(* IEC 61131-3 sources: beckhoffAutomationInterface/ST/Shark/App/Shark/Programs, 13 files *)

(* ---- PRG_BronkhorstPressure.st ---- *)
(* Bronkhorst pressure controller application (Modbus needle valves).
   Creates Modbus hardware stack and controllers, then injects
   controller interfaces into PRG_PRESSURE_SENSOR via Configure(). *)
PROGRAM PRG_BronkhorstPressure
VAR
    // Modbus Hardware Stack
    fbModbusMaster       : ModbusRtuMasterV2_KL6x22B;
    fbNetworkCoordinator : FB_ModbusNetworkCoordinator;

    // Per-controller hardware
    aHardwareHandlers : ARRAY[1..GVL_PressureSystem.CONTROLLER_COUNT] OF FB_ModbusHardwareHandler;
    aDrivers          : ARRAY[1..GVL_PressureSystem.CONTROLLER_COUNT] OF FB_BronkhorstModbusAdapter;

    // Controllers
    aControllers : ARRAY[1..GVL_PressureSystem.CONTROLLER_COUNT] OF FB_BronkhorstController;
    aInterfaces  : ARRAY[1..GVL_PressureSystem.CONTROLLER_COUNT] OF I_Controller;

    bInitialized : BOOL := FALSE;
    i : INT;
END_VAR

    IF NOT bInitialized THEN
        _Init();
    END_IF

    // Execute Modbus communication
    fbModbusMaster();
    fbNetworkCoordinator.Execute();

    // Execute controllers
    FOR i := 1 TO GVL_PressureSystem.CONTROLLER_COUNT DO
        aControllers[i].Execute();
    END_FOR

METHOD PRIVATE _Init
    // PrecursorHot (slave 1)
    _InitController(
        eId           := E_PressureController.A_Side,
        nSlaveAddress := GVL_PressureSystem.MODBUS_FIRST_SLAVE_ADDRESS
    );

    // ReactantHot (slave 2)
    _InitController(
        eId           := E_PressureController.B_Side,
        nSlaveAddress := GVL_PressureSystem.MODBUS_FIRST_SLAVE_ADDRESS + 1
    );

    fbNetworkCoordinator.Init();

    // Inject controllers into pressure subsystem
    PRG_PRESSURE_SENSOR.Configure(aipCtrl := aInterfaces);

    bInitialized := TRUE;
END_METHOD

METHOD PRIVATE _InitController
VAR_INPUT
    eId           : E_PressureController;
    nSlaveAddress : BYTE;
END_VAR
VAR
    nIdx : INT;
END_VAR
    nIdx := eId;

    aHardwareHandlers[nIdx].Init(
        sInstanceName    := CONCAT('MODBUS_PRES_', TO_STRING(eId)),
        pModbusRtuMaster := ADR(fbModbusMaster),
        nSlaveAddress    := nSlaveAddress
    );
    aDrivers[nIdx].Init(
        sInstanceName      := CONCAT('DRV_', TO_STRING(eId)),
        nSlaveAddress      := nSlaveAddress,
        ipModbusComm       := aHardwareHandlers[nIdx],
        rFullScaleCapacity := GVL_PressureSystem.MAX_PRESSURE_CTRL_BAR,
        rMinimumValue      := GVL_PressureSystem.MIN_PRESSURE_CTRL_BAR
    );

    fbNetworkCoordinator.AddSlave(aDrivers[nIdx]);
    aDrivers[nIdx].SetPIDMode();

    aControllers[nIdx].Init(
        sInstanceName      := TO_STRING(eId),
        ipHardware         := aDrivers[nIdx],
        rMinValue          := GVL_PressureSystem.MIN_PRESSURE_CTRL_BAR,
        rMaxValue          := GVL_PressureSystem.MAX_PRESSURE_CTRL_BAR,
        bInverseControl    := TRUE,
        rBoundaryTolerance := GVL_PressureSystem.SETPOINT_TOLERANCE
    );

    aInterfaces[nIdx] := aControllers[nIdx];
END_METHOD

END_PROGRAM

(* ---- PRG_DIGITAL_INPUT.st ---- *)
(*
Digital Input Program - Shark System
Manages all digital inputs with centralized initialization.
*)
PROGRAM PRG_DIGITAL_INPUT
VAR
    // Subsystem and Manual Panel
    fbDigitalInputSubsystem : FB_DigitalInputSubsystem;
    fbManualPanel           : FB_DigitalInputManualPanel;

    // Hardware IO - Door Proximity Sensors
    IO_DoorLT            AT %I* : BOOL;
    IO_DoorLM            AT %I* : BOOL;
    IO_DoorLB            AT %I* : BOOL;
    IO_DoorRT            AT %I* : BOOL;
    IO_DoorRM            AT %I* : BOOL;
    IO_DoorRB            AT %I* : BOOL;
    IO_DoorBML           AT %I* : BOOL;
    IO_DoorBMR           AT %I* : BOOL;
    IO_DoorBMB           AT %I* : BOOL;

    // Safety-derived digital inputs (logical, not physical IO).
    // Updated each cycle from FB_SafetyManager via Configure()/I_SafetyStatus.
    _bHeaterVoltOn   : BOOL := FALSE;  // HETR_VOLT_ON — HeaterVoltagePresence
    _bSafetyOk       : BOOL := FALSE;  // SAFE_STO_ON  — safety state machine OK
    _bSafetyOverride : BOOL := TRUE;   // SAFE_OVERRIDE — no physical switch on Shark; always active

    // Safety status interface (injected via Configure)
    _ipSafety : I_SafetyStatus;

    // Function blocks and interfaces
    afbInputs : ARRAY[1..GVL_DIOConfig.DI_COUNT] OF FB_DigitalInput;
    aipInputs : ARRAY[1..GVL_DIOConfig.DI_COUNT] OF I_DigitalInput;

    bInitialized : BOOL := FALSE;
END_VAR

    IF NOT bInitialized THEN
        _Init();
    END_IF

    // Refresh safety-derived inputs before Execute() so subsystem reads fresh values each scan
    IF _ipSafety <> 0 THEN
        _bHeaterVoltOn := _ipSafety.HeaterVoltagePresence;
        _bSafetyOk     := _ipSafety.IsOk;
        // _bSafetyOverride stays TRUE — Shark has no physical override switch
    END_IF

    fbDigitalInputSubsystem.Execute();
    fbManualPanel(ipSubsystem := fbDigitalInputSubsystem, nMaxInput := GVL_DIOConfig.DI_COUNT);

METHOD PRIVATE _Init
VAR
    i : INT;
    apIO : ARRAY[1..GVL_DIOConfig.DI_COUNT] OF POINTER TO BOOL;
END_VAR
    // Build IO pointer mapping
    apIO[E_DigitalInputIdentifier.PRXS_DOOR_LT]    := ADR(IO_DoorLT);
    apIO[E_DigitalInputIdentifier.PRXS_DOOR_LM]    := ADR(IO_DoorLM);
    apIO[E_DigitalInputIdentifier.PRXS_DOOR_LB]    := ADR(IO_DoorLB);
    apIO[E_DigitalInputIdentifier.PRXS_DOOR_RT]    := ADR(IO_DoorRT);
    apIO[E_DigitalInputIdentifier.PRXS_DOOR_RM]    := ADR(IO_DoorRM);
    apIO[E_DigitalInputIdentifier.PRXS_DOOR_RB]    := ADR(IO_DoorRB);
    apIO[E_DigitalInputIdentifier.PRXS_DOOR_BML]   := ADR(IO_DoorBML);
    apIO[E_DigitalInputIdentifier.PRXS_DOOR_BMR]   := ADR(IO_DoorBMR);
    apIO[E_DigitalInputIdentifier.PRXS_DOOR_BMB]   := ADR(IO_DoorBMB);
    apIO[E_DigitalInputIdentifier.HETR_VOLT_ON]  := ADR(_bHeaterVoltOn);
    apIO[E_DigitalInputIdentifier.SAFE_STO_ON]   := ADR(_bSafetyOk);
    apIO[E_DigitalInputIdentifier.SAFE_OVERRIDE] := ADR(_bSafetyOverride);

    // Initialize all inputs using the mapping (all N.O. sensors, no inversion needed)
    FOR i := 1 TO GVL_DIOConfig.DI_COUNT DO
        IF apIO[i] <> 0 THEN
            afbInputs[i].Init(INT_TO_STRING(i), apIO[i]^);
            aipInputs[i] := afbInputs[i];
        END_IF
    END_FOR

    fbDigitalInputSubsystem.Init(aipInputs := aipInputs, nCount := GVL_DIOConfig.DI_COUNT);
    bInitialized := TRUE;
END_METHOD

METHOD PUBLIC Init : BOOL
VAR_INPUT
    ipSafety : I_SafetyStatus;
END_VAR
    IF ipSafety = 0 THEN
        Init := FALSE;
        RETURN;
    END_IF
    _ipSafety := ipSafety;
    Init := TRUE;
END_METHOD

END_PROGRAM

(* ---- PRG_DIGITAL_OUTPUT.st ---- *)
(*
Digital Output Program - Shark System
Manages all digital outputs with centralized initialization.
*)
PROGRAM PRG_DIGITAL_OUTPUT
VAR
    // Subsystem and Manual Panel
    fbDigitalOutputSubsystem : FB_DigitalOutputSubsystem;
    fbManualPanel            : FB_DigitalOutputManualPanel;

    // Hardware IO (Digital Outputs) - Signal Lights
    IO_SignalRed         AT %Q* : BOOL;
    IO_SignalYellow      AT %Q* : BOOL;
    IO_SignalGreen       AT %Q* : BOOL;

    // Hardware IO - Camera Lights
    IO_CameraLightTop    AT %Q* : BOOL;
    IO_CameraLightSide   AT %Q* : BOOL;

    // Hardware IO - Vacuum Pumps
    IO_ExhaustPump       AT %Q* : BOOL;
    IO_ChuckVacuumPump   AT %Q* : BOOL;

    // Hardware IO - Chiller
    IO_ChillerPower      AT %Q* : BOOL;

    // Hardware IO - Door Locks
    IO_DoorLockFL        AT %Q* : BOOL;
    IO_DoorLockFR        AT %Q* : BOOL;

    // Hardware IO - Heater Voltage Enable
    IO_HeaterVoltageOn   AT %Q* : BOOL;

    // Hardware IO - Solenoid Valve Outputs (consumed by PRG_VALVE)
    IO_ChuckLZ1          AT %Q* : BOOL;
    IO_ChuckLZ2          AT %Q* : BOOL;
    IO_ChuckLZ3          AT %Q* : BOOL;
    IO_ChuckVent         AT %Q* : BOOL;
    IO_ChuckWaterIn      AT %Q* : BOOL;
    IO_ChuckWaterOut     AT %Q* : BOOL;

    // Function blocks and interfaces
    afbOutputs : ARRAY[1..GVL_DIOConfig.DO_COUNT] OF FB_DigitalOutput;
    aipOutputs : ARRAY[1..GVL_DIOConfig.DO_COUNT] OF I_DigitalOutput;

    bInitialized : BOOL := FALSE;
END_VAR

    IF NOT bInitialized THEN
        _Init();
    END_IF

    fbDigitalOutputSubsystem.Execute();
    fbManualPanel(ipSubsystem := fbDigitalOutputSubsystem, nMaxOutput := GVL_DIOConfig.DO_COUNT);

METHOD PRIVATE _Init
VAR
    i : INT;
    apIO       : ARRAY[1..GVL_DIOConfig.DO_COUNT] OF POINTER TO BOOL;
    aSafeState : ARRAY[1..GVL_DIOConfig.DO_COUNT] OF BOOL;
END_VAR
    // ------------------------------------------------------------------
    // Safe states — applied by SetSafeState() on sequence abort / Halt().
    // Every output that is not listed here defaults to FALSE (de-energise).
    // SAFETY: door locks TRUE = stay locked; chiller TRUE = keep running.
    // ------------------------------------------------------------------
    aSafeState[E_DigitalOutputIdentifier.PUMP_AB_EXH]   := TRUE;
    aSafeState[E_DigitalOutputIdentifier.LGHT_SGN_GRN]  := FALSE; // Lights off
    aSafeState[E_DigitalOutputIdentifier.LGHT_SGN_RED]  := FALSE;
    aSafeState[E_DigitalOutputIdentifier.LGHT_SGN_YEL]  := FALSE;
    aSafeState[E_DigitalOutputIdentifier.LGHT_CMR_TOP]  := TRUE;
    aSafeState[E_DigitalOutputIdentifier.LGHT_CMR_SIDE] := TRUE;
    aSafeState[E_DigitalOutputIdentifier.CHIL_PWR]      := TRUE;  // SAFETY: chiller must keep running to protect hardware
    aSafeState[E_DigitalOutputIdentifier.LOCK_DOOR_FL]  := TRUE;  // SAFETY: doors stay locked on abort
    aSafeState[E_DigitalOutputIdentifier.LOCK_DOOR_FR]  := TRUE;  // SAFETY: doors stay locked on abort
    aSafeState[E_DigitalOutputIdentifier.VALV_CHK_LZ1]  := FALSE; // Chuck zone valves close
    aSafeState[E_DigitalOutputIdentifier.VALV_CHK_LZ2]  := FALSE;
    aSafeState[E_DigitalOutputIdentifier.VALV_CHK_LZ3]  := FALSE;
    aSafeState[E_DigitalOutputIdentifier.VALV_CHK_VENT] := FALSE; // Vent closes
    aSafeState[E_DigitalOutputIdentifier.VALV_CHK_WIN]  := FALSE; // Water valves close
    aSafeState[E_DigitalOutputIdentifier.VALV_CHK_WOUT] := FALSE;

    // Build IO pointer mapping
    apIO[E_DigitalOutputIdentifier.LGHT_SGN_RED]   := ADR(IO_SignalRed);
    apIO[E_DigitalOutputIdentifier.LGHT_SGN_YEL]   := ADR(IO_SignalYellow);
    apIO[E_DigitalOutputIdentifier.LGHT_SGN_GRN]   := ADR(IO_SignalGreen);
    apIO[E_DigitalOutputIdentifier.LGHT_CMR_TOP]   := ADR(IO_CameraLightTop);
    apIO[E_DigitalOutputIdentifier.LGHT_CMR_SIDE]  := ADR(IO_CameraLightSide);
    apIO[E_DigitalOutputIdentifier.PUMP_AB_EXH]    := ADR(IO_ExhaustPump);
    apIO[E_DigitalOutputIdentifier.PUMP_CHK_VAC]   := ADR(IO_ChuckVacuumPump);
    apIO[E_DigitalOutputIdentifier.CHIL_PWR]       := ADR(IO_ChillerPower);
    apIO[E_DigitalOutputIdentifier.LOCK_DOOR_FL]   := ADR(IO_DoorLockFL);
    apIO[E_DigitalOutputIdentifier.LOCK_DOOR_FR]   := ADR(IO_DoorLockFR);
    apIO[E_DigitalOutputIdentifier.VALV_CHK_LZ1]   := ADR(IO_ChuckLZ1);
    apIO[E_DigitalOutputIdentifier.VALV_CHK_LZ2]   := ADR(IO_ChuckLZ2);
    apIO[E_DigitalOutputIdentifier.VALV_CHK_LZ3]   := ADR(IO_ChuckLZ3);
    apIO[E_DigitalOutputIdentifier.VALV_CHK_VENT]  := ADR(IO_ChuckVent);
    apIO[E_DigitalOutputIdentifier.VALV_CHK_WIN]   := ADR(IO_ChuckWaterIn);
    apIO[E_DigitalOutputIdentifier.VALV_CHK_WOUT]  := ADR(IO_ChuckWaterOut);

    // Initialize all outputs using the mapping
    FOR i := 1 TO GVL_DIOConfig.DO_COUNT DO
        IF apIO[i] <> 0 THEN
            afbOutputs[i].Init(INT_TO_STRING(i), apIO[i]^, aSafeState[i]);
            aipOutputs[i] := afbOutputs[i];
        END_IF
    END_FOR

    fbDigitalOutputSubsystem.Init(aipOutputs := aipOutputs, nCount := GVL_DIOConfig.DO_COUNT);
    bInitialized := TRUE;
END_METHOD

END_PROGRAM

(* ---- PRG_HEAT_ZONE.st ---- *)
PROGRAM PRG_HEAT_ZONE
(*
Shark heater output wiring + temperature subsystem entry point.

  * 10 SSR outputs (one per channel) split across 8 zones.
  * Channel ordering MUST match PRG_TEMPERATURE_SENSOR's channel layout.
*)
VAR
    // --- Heater Digital Outputs (linked to EtherCAT process image) ---
    // HETR_HEAD   (channel 1)
    HEAD_Htr          AT %Q* : BOOL;
    // HETR_A_STR  (channel 2)
    A_STR_Htr         AT %Q* : BOOL;
    // HETR_A_CMB  (channel 3)
    A_CMB_Htr         AT %Q* : BOOL;
    // HETR_A_B1   (channel 4)
    A_B1_Htr          AT %Q* : BOOL;
    // HETR_A_B2   (channel 5)
    A_B2_Htr          AT %Q* : BOOL;
    // HETR_A_B3   (channel 6)
    A_B3_Htr          AT %Q* : BOOL;
    // HETR_B_STR  (channel 7)
    B_STR_Htr         AT %Q* : BOOL;
    // HETR_B_CMB  (channel 8)
    B_CMB_Htr         AT %Q* : BOOL;
    // HETR_B_B1   (channel 9)
    B_B1_Htr          AT %Q* : BOOL;
    // HETR_B_B2   (channel 10)
    B_B2_Htr          AT %Q* : BOOL;
    // HETR_B_B3   (channel 11)
    B_B3_Htr          AT %Q* : BOOL;
    // HETR_EXH    (channels 12..13)
    EXH_Htr           AT %Q* : BOOL;
    EXH_E2_Htr        AT %Q* : BOOL;
    // HETR_CHK    (channels 14..15)
    CHK_Htr           AT %Q* : BOOL;
    CHK_E2_Htr        AT %Q* : BOOL;

    // --- Heater Adapters ---
    afbElementHeaters : ARRAY[1..GVL_TemperatureZones.CHANNEL_MAX] OF FB_DigitalOutput;

    // --- Interface array consumed by FB_TemperatureSubsystem ---
    aipChannelHeaters : ARRAY[1..GVL_TemperatureZones.CHANNEL_MAX] OF I_DigitalOutput;

    // --- Application ---
    fbTemperatureSubsystem : FB_TemperatureSubsystem;
    fbManualPanel          : FB_TemperatureManualPanel;
    fbTuningPanel          : FB_BeckhoffTuningPanel;

    bInitialized : BOOL := FALSE;
END_VAR

    IF NOT bInitialized THEN
        _Init();
    END_IF

    // Run all zones and channels
    fbTemperatureSubsystem.Execute();

    // HMI Panels
    fbManualPanel(ipSubsystem := fbTemperatureSubsystem, nMaxZone := GVL_TemperatureZones.CONTROLLABLE_ZONE_MAX);
    fbTuningPanel(
        ipTunable := fbTemperatureSubsystem.GetTunable(
            eZone       := fbTuningPanel.iSelectedZoneIdx,
            nChannelIdx := fbTuningPanel.iSelectedChannelIdx,
            bWholeZone  := fbTuningPanel.bTuneWholeZone)
    );

METHOD PRIVATE _Init
    // Initialize channel heaters in channel-order (matches PRG_TEMPERATURE_SENSOR).
    _InitElement(1,  HEAD_Htr);
    _InitElement(2,  A_STR_Htr);
    _InitElement(3,  A_CMB_Htr);
    _InitElement(4,  A_B1_Htr);
    _InitElement(5,  A_B2_Htr);
    _InitElement(6,  A_B3_Htr);
    _InitElement(7,  B_STR_Htr);
    _InitElement(8,  B_CMB_Htr);
    _InitElement(9,  B_B1_Htr);
    _InitElement(10, B_B2_Htr);
    _InitElement(11, B_B3_Htr);
    _InitElement(12, EXH_Htr);
    _InitElement(13, EXH_E2_Htr);
    _InitElement(14, CHK_Htr);
    _InitElement(15, CHK_E2_Htr);

    // Initialize subsystem (sensors come from PRG_TEMPERATURE_SENSOR)
    bInitialized := fbTemperatureSubsystem.Init(
        aipChannelSensors := PRG_TEMPERATURE_SENSOR.aipChannelSensors,
        aipMonitorSensors := PRG_TEMPERATURE_SENSOR.aipMonitorSensors,
        aipChannelHeaters := aipChannelHeaters
    );
END_METHOD

METHOD PRIVATE _InitElement
VAR_INPUT
    nGlobalIdx : INT;
END_VAR
VAR_IN_OUT
    bOutput : BOOL;
END_VAR
    afbElementHeaters[nGlobalIdx].Init(
        sInstanceName := CONCAT('HEATER_E', TO_STRING(nGlobalIdx)),
        ipOutputRef   := bOutput
    );
    aipChannelHeaters[nGlobalIdx] := afbElementHeaters[nGlobalIdx];
END_METHOD

END_PROGRAM

(* ---- PRG_HUMIDITY_SENSOR.st ---- *)
(*
PRG_HUMIDITY_SENSOR — Ambient Humidity Sensor (Shark)

Manages the MDP5001_300_7E2119CA humidity channel from the Shark TH sensor pair.
Consumers read the scaled value via ipSensor.GetMeasurement().

The temperature channel of the same TH sensor is wired in PRG_TEMPERATURE_SENSOR
as E_TemperatureMonitorZone.SENS_CHAMBER.

Scaling constants are in GVL_HumiditySystem.
*)
PROGRAM PRG_HUMIDITY_SENSOR
VAR_INPUT
    // Hardware IO — linked to EtherCAT process image at %I* offset matching terminal position.
    // VAR_INPUT allows PRG_SIMULATION to write raw values for simulation mode.
    IO_Humid : T_Beckhoff_AmbientSensor;
END_VAR
VAR
    fbAdapter    : FB_AnalogInputAdapter;
    fbSensor     : FB_AnalogSensor;
    ipSensor     : I_Sensor;
    bInitialized : BOOL := FALSE;
END_VAR

    IF NOT bInitialized THEN
        _Init();
    END_IF

    fbAdapter.Execute();
    fbSensor.Execute();

METHOD PRIVATE _Init
    fbAdapter.Link(ADR(IO_Humid));
    fbSensor.Init(
        sInstanceName := 'AMBT_HUMID',
        ipRawInput    := fbAdapter,
        rRawMin       := GVL_HumiditySystem.AMBT_HUMID_RAW_MIN,
        rRawMax       := GVL_HumiditySystem.AMBT_HUMID_RAW_MAX,
        rScaledMin    := GVL_HumiditySystem.AMBT_HUMID_SCALED_MIN,
        rScaledMax    := GVL_HumiditySystem.AMBT_HUMID_SCALED_MAX
    );
    ipSensor     := fbSensor;
    bInitialized := TRUE;
END_METHOD

END_PROGRAM

(* ---- PRG_MFC.st ---- *)
PROGRAM PRG_MFC
VAR
    // Hardware IO - MFC Controllers (Bronkhorst EtherCAT)
    // Declared as VAR (not VAR_INPUT) so TwinCAT I/O linker exposes AT %I*/%Q*
    // members for EtherCAT PDO mapping. PRG_SIMULATION writes to these directly
    // via PRG_MFC.IO_MFC_*.MeasuredValue — this works identically for VAR.
    IO_MFC_Precursor : ST_BronkhorstController_IO;  // Range: 0-25 sccm
    IO_MFC_Reactant  : ST_BronkhorstController_IO;  // Range: 0-25 sccm
    IO_MFC_Inert     : ST_BronkhorstController_IO;  // Range: 0-500 sccm
END_VAR
VAR
    // Subsystem and Manual Panel
    fbFlowSubsystem : FB_FlowSubsystem;
    fbManualPanel   : FB_FlowManualPanel;

    // Adapters
    adapterPrecursor : FB_BronkhorstEtherCATAdapter;
    adapterReactant  : FB_BronkhorstEtherCATAdapter;
    adapterInert     : FB_BronkhorstEtherCATAdapter;

    // Controllers
    mfcPrecursor : FB_BronkhorstController;
    mfcReactant  : FB_BronkhorstController;
    mfcInert     : FB_BronkhorstController;

    bInitialized : BOOL := FALSE;
END_VAR

    IF NOT bInitialized THEN
        _Init();
    END_IF

    // Execute Controllers
    mfcPrecursor.Execute();
    mfcReactant.Execute();
    mfcInert.Execute();

    // Execute Subsystem (Error Aggregation)
    fbFlowSubsystem.Execute();

    // Manual Panel
    fbManualPanel(ipSubsystem := fbFlowSubsystem, nMaxZone := GVL_FlowSystem.FLOW_ZONE_COUNT);

METHOD PRIVATE _Init
VAR
    aipControllers : ARRAY[1..GVL_FlowSystem.FLOW_ZONE_COUNT] OF I_Controller;
END_VAR
    _InitMfc(
        eId          := E_MFCIdentifier.MFCT_A_01,
        stIo         := IO_MFC_Precursor,
        fbAdapter    := adapterPrecursor,
        fbController := mfcPrecursor,
        rMinValue    := GVL_FlowSystem.MIN_FLOW_PRECURSOR_SCCM,
        rMaxValue    := GVL_FlowSystem.MAX_FLOW_PRECURSOR_SCCM
    );
    _InitMfc(
        eId          := E_MFCIdentifier.MFCT_B_01,
        stIo         := IO_MFC_Reactant,
        fbAdapter    := adapterReactant,
        fbController := mfcReactant,
        rMinValue    := GVL_FlowSystem.MIN_FLOW_REACTANT_SCCM,
        rMaxValue    := GVL_FlowSystem.MAX_FLOW_REACTANT_SCCM
    );
    _InitMfc(
        eId          := E_MFCIdentifier.MFCT_IG_01,
        stIo         := IO_MFC_Inert,
        fbAdapter    := adapterInert,
        fbController := mfcInert,
        rMinValue    := GVL_FlowSystem.MIN_FLOW_INERT_SCCM,
        rMaxValue    := GVL_FlowSystem.MAX_FLOW_INERT_SCCM
    );

    // Subsystem Initialization
    aipControllers[E_MFCIdentifier.MFCT_A_01]  := mfcPrecursor;
    aipControllers[E_MFCIdentifier.MFCT_B_01]  := mfcReactant;
    aipControllers[E_MFCIdentifier.MFCT_IG_01] := mfcInert;

    fbFlowSubsystem.Init(aipControllers := aipControllers, nCount := GVL_FlowSystem.FLOW_ZONE_COUNT);
    bInitialized := TRUE;
END_METHOD

METHOD PRIVATE _InitMfc
VAR_INPUT
    eId       : E_MFCIdentifier;
    rMinValue : REAL;
    rMaxValue : REAL;
END_VAR
VAR_IN_OUT
    stIo         : ST_BronkhorstController_IO;
    fbAdapter    : FB_BronkhorstEtherCATAdapter;
    fbController : FB_BronkhorstController;
END_VAR
    fbAdapter.Link(
        refMeasuredValue     := stIo.MeasuredValue,
        refActualSetpoint    := stIo.ActualSetpoint,
        refValveOutput       := stIo.ValveOutput,
        refCommandedSetpoint := stIo.CommandedSetpoint,
        refControlByte       := stIo.ControlByte,
        refControlMode       := stIo.ControlMode,
        rMinValue            := REAL_TO_LREAL(rMinValue),
        rMaxValue            := REAL_TO_LREAL(rMaxValue)
    );
    fbController.Init(
        sInstanceName      := TO_STRING(eId),
        ipHardware         := fbAdapter,
        rMinValue          := rMinValue,
        rMaxValue          := rMaxValue,
        bInverseControl    := FALSE,
        rBoundaryTolerance := GVL_FlowSystem.SETPOINT_TOLERANCE
    );
END_METHOD

END_PROGRAM

(* ---- PRG_PRESSURE_SENSOR.st ---- *)
(*
Pressure Sensor Program - Shark System
Manages 4 analog pressure sensors with per-sensor scaling.
Bronkhorst pressure controllers are managed by PRG_BronkhorstPressure
and injected via Configure().

NOTE: PSNS_CHK_VAC has inverted physical mapping (higher raw = more vacuum = lower pressure).
      FB_AnalogSensor requires ascending ranges, so the reading is physically inverted.
      Consumers must compute: actual_pressure_bar = 1.0165 - sensor_reading
      TODO: Consider extending FB_AnalogSensor to support inverted scaling.
*)
PROGRAM PRG_PRESSURE_SENSOR
VAR
    // Hardware IO - Analog Pressure Sensors
    // Declared as VAR (not VAR_INPUT) so TwinCAT I/O linker exposes AT %I*/%Q*
    // members for EtherCAT PDO mapping. PRG_SIMULATION writes to these via
    // pointer/ADR — this works identically for VAR.
    IO_PressureSensors : ARRAY[1..GVL_PressureSystem.SENSOR_COUNT] OF T_Beckhoff_PressureSensor;
END_VAR
VAR
    // Subsystem and Manual Panel
    fbPressureSubsystem : FB_PressureSubsystem;
    fbManualPanel       : FB_PressureManualPanel;

    // Adapters and Sensors
    afbAdapters : ARRAY[1..GVL_PressureSystem.SENSOR_COUNT] OF FB_AnalogInputAdapter;
    afbSensors  : ARRAY[1..GVL_PressureSystem.SENSOR_COUNT] OF FB_AnalogSensor;

    // Interface arrays
    aipSensors     : ARRAY[1..GVL_PressureSystem.SENSOR_COUNT] OF I_Sensor;
    aipControllers : ARRAY[1..GVL_PressureSystem.CONTROLLER_COUNT] OF I_Controller;

    bConfigured     : BOOL := FALSE;
    bInitialized    : BOOL := FALSE;
    _bNotConfiguredLogged : BOOL := FALSE;
    i : INT;
END_VAR

    IF NOT bConfigured THEN
        IF NOT _bNotConfiguredLogged THEN
            GVL_ErrorLogger.Logger.LogError(
                sSource  := 'PRG_PRESSURE_SENSOR',
                eErrorId := E_ErrorId.ERR_GEN_NOT_CONFIGURED,
                sContext := 'PRG_PRESSURE_SENSOR executed before Configure(); pressure sensors will not run'
            );
            _bNotConfiguredLogged := TRUE;
        END_IF
        RETURN;
    END_IF

    IF NOT bInitialized THEN
        _Init();
    END_IF

    // Execute adapters and sensors
    FOR i := 1 TO GVL_PressureSystem.SENSOR_COUNT DO
        afbAdapters[i].Execute();
        afbSensors[i].Execute();
    END_FOR

    // Execute subsystem (error aggregation)
    fbPressureSubsystem.Execute();
    fbManualPanel(ipSubsystem := fbPressureSubsystem, nMaxSensor := GVL_PressureSystem.SENSOR_COUNT, nMaxCtrl := GVL_PressureSystem.CONTROLLER_COUNT);

    // Dependency injection - accepts controller interfaces from PRG_BronkhorstPressure
METHOD PUBLIC Configure
VAR_INPUT
    aipCtrl : ARRAY[1..GVL_PressureSystem.CONTROLLER_COUNT] OF I_Controller;
END_VAR
VAR
    iLocal : INT;
END_VAR
    IF bConfigured THEN RETURN;
    END_IF

    FOR iLocal := 1 TO GVL_PressureSystem.CONTROLLER_COUNT DO
        aipControllers[iLocal] := aipCtrl[iLocal];
    END_FOR

    bConfigured := TRUE;
END_METHOD

METHOD PRIVATE _Init
VAR
    eId : E_PressureSensorIdentifier;
END_VAR
    // PSNS_A_DST: A-side Distributor [0-3 bar]
    _InitSensor(
        eId       := E_PressureSensorIdentifier.PSNS_A_DST,
        rRawMin   := GVL_PressureSystem.PSNS_A_DST_RAW_MIN,
        rRawMax   := GVL_PressureSystem.PSNS_A_DST_RAW_MAX,
        rScaledMin := GVL_PressureSystem.PSNS_A_DST_SCALED_MIN,
        rScaledMax := GVL_PressureSystem.PSNS_A_DST_SCALED_MAX
    );

    // PSNS_B_DST: B-side Distributor [0-3 bar]
    _InitSensor(
        eId       := E_PressureSensorIdentifier.PSNS_B_DST,
        rRawMin   := GVL_PressureSystem.PSNS_B_DST_RAW_MIN,
        rRawMax   := GVL_PressureSystem.PSNS_B_DST_RAW_MAX,
        rScaledMin := GVL_PressureSystem.PSNS_B_DST_SCALED_MIN,
        rScaledMax := GVL_PressureSystem.PSNS_B_DST_SCALED_MAX
    );

    // PSNS_AB_EXH: Exhaust Vacuum [0-1 bar]
    _InitSensor(
        eId       := E_PressureSensorIdentifier.PSNS_AB_EXH,
        rRawMin   := GVL_PressureSystem.PSNS_AB_EXH_RAW_MIN,
        rRawMax   := GVL_PressureSystem.PSNS_AB_EXH_RAW_MAX,
        rScaledMin := GVL_PressureSystem.PSNS_AB_EXH_SCALED_MIN,
        rScaledMax := GVL_PressureSystem.PSNS_AB_EXH_SCALED_MAX
    );

    // PSNS_CHK_VAC: Chuck Vacuum [inverted: see NOTE above]
    _InitSensor(
        eId       := E_PressureSensorIdentifier.PSNS_CHK_VAC,
        rRawMin   := GVL_PressureSystem.PSNS_CHK_VAC_RAW_MIN,
        rRawMax   := GVL_PressureSystem.PSNS_CHK_VAC_RAW_MAX,
        rScaledMin := GVL_PressureSystem.PSNS_CHK_VAC_SCALED_MIN,
        rScaledMax := GVL_PressureSystem.PSNS_CHK_VAC_SCALED_MAX
    );

    // Initialize subsystem with sensors + injected controllers
    fbPressureSubsystem.Init(aipSensors := aipSensors, nSensorCount := GVL_PressureSystem.SENSOR_COUNT, aipControllers := aipControllers, nControllerCount := GVL_PressureSystem.CONTROLLER_COUNT);
    bInitialized := TRUE;
END_METHOD

METHOD PRIVATE _InitSensor
VAR_INPUT
    eId        : E_PressureSensorIdentifier;
    rRawMin    : LREAL;
    rRawMax    : LREAL;
    rScaledMin : LREAL;
    rScaledMax : LREAL;
END_VAR
VAR
    nIdx : INT;
END_VAR
    nIdx := eId;

    afbAdapters[nIdx].Link(ADR(IO_PressureSensors[nIdx]));
    afbSensors[nIdx].Init(
        sInstanceName := TO_STRING(eId),
        ipRawInput    := afbAdapters[nIdx],
        rRawMin       := rRawMin,
        rRawMax       := rRawMax,
        rScaledMin    := rScaledMin,
        rScaledMax    := rScaledMax
    );
    aipSensors[nIdx] := afbSensors[nIdx];
END_METHOD

END_PROGRAM

(* ---- PRG_Sequence.st ---- *)
// Runs the sequence orchestrator and the sequence tester side-by-side.
// Tester is wired to the orchestrator during Configure — no separate PRG_SequenceTester needed.
PROGRAM PRG_Sequence
VAR
    fbOrchestrator : FB_SequenceOrchestrator;
    fbTester       : FB_SequenceTester;
END_VAR

    fbOrchestrator();
    fbTester();

END_PROGRAM

METHOD PUBLIC Configure : BOOL
VAR_INPUT
    ipProvider : I_HardwareProvider;
END_VAR
    Configure := fbOrchestrator.Configure(ipProvider := ipProvider);
    fbTester.Configure(refOrchestrator := fbOrchestrator);
END_METHOD

METHOD PUBLIC GetStatus : ST_SequenceStatus
    GetStatus := fbOrchestrator.GetStatus();
END_METHOD

(* ---- PRG_SIMULATION.st ---- *)
(*
PRG_SIMULATION — I/O Hijacking Simulator for Shark Machine

Writes directly to the bottom-most layer:
  - Beckhoff sensor structs (T_Beckhoff_TempSensor_*, T_Beckhoff_PressureSensor)
    via raw INT pointer writes at offset 2.
  - Bronkhorst Modbus adapters via InjectMeasuredValue() (overwrites the polled
    rMeasuredValue, symmetric to PRO's EtherCAT IO struct hijack).
  - EtherCAT MFC IO fields (ST_BronkhorstController_IO.MeasuredValue) directly.

Everything above (FB_AnalogInputAdapter → FB_AnalogSensor → controllers → UI)
works naturally without knowing it's simulated.

Shark has 10 heater zones (no B-side zones 7-11), 4 pressure sensors,
3 EtherCAT MFCs, and Modbus-based pressure controllers.

PHYSICS ENGINE:
  FB_GasPhysicsSimulator reads valve states + pump state from the previous cycle,
  computes CM/HM pressures and MFC flow, and outputs are written to sensor IO.
*)
PROGRAM PRG_SIMULATION
VAR
    // Hardware provider — injected via Configure() from PRG_SHARK
    _ipProvider  : I_HardwareProvider;
    _bConfigured : BOOL := FALSE;

    // Gas system physics — pressure + flow for both sides
    fbGasPhysics : FB_GasPhysicsSimulator;

    // Temperature physics — one per channel channel
    aSimHeaters : ARRAY[1..GVL_TemperatureZones.CHANNEL_MAX] OF FB_SimulateHeaterZone;

    // Inert MFC simulation (not part of gas side physics)
    fbSimMFC_Inert : FB_SimulateAnalogActuator;

    // Working
    bInitialized : BOOL := FALSE;
END_VAR

IF NOT GVL_Simulation.bActive THEN
    RETURN;
END_IF

IF NOT bInitialized THEN
    _Init();
END_IF

// =============================================================================
// 0. SAFETY — Force safe state so subsystems can run
// =============================================================================
GVL_Safety.SafetyOk := TRUE;
GVL_Safety.HeaterVoltage := 230.0;

// =============================================================================
// 1. TEMPERATURE — Write directly to T_Beckhoff_TempSensor structs (no provider)
// =============================================================================
_SimulateTemperature();

// =============================================================================
// 2. GAS PHYSICS + PRESSURE + MFC (requires provider — first cycle is a no-op,
//    _Init atmospheric seed is preserved until provider is wired on cycle 2)
// =============================================================================
IF _bConfigured THEN
    _SimulateGasPhysics();
    _SimulatePressureSensors();
    _SimulateMFCs();
    _SimulateModbusPressureControllers();
END_IF

// =============================================================================
// CONFIGURATION
// =============================================================================

METHOD PUBLIC Configure
VAR_INPUT
    ipProvider : I_HardwareProvider;
END_VAR
    _ipProvider  := ipProvider;
    _bConfigured := _ipProvider <> 0;
END_METHOD

// =============================================================================
// INITIALIZATION
// =============================================================================

METHOD PRIVATE _Init
VAR
    iZone      : INT;
    e          : INT;
    nGlobalIdx : INT;
    nCount     : INT;
    iSensor    : INT;
END_VAR
    // Temperature: init physics for every channel of every populated zone
    nGlobalIdx := 0;
    FOR iZone := 1 TO GVL_TemperatureZones.CONTROLLABLE_ZONE_MAX DO
        nCount := GVL_TemperatureZoneConfig.ZONE_CONFIG[iZone].nChannelCount;
        FOR e := 1 TO nCount DO
            nGlobalIdx := nGlobalIdx + 1;
            IF nGlobalIdx > GVL_TemperatureZones.CHANNEL_MAX THEN EXIT; END_IF
            IF GVL_TemperatureZoneConfig.ZONE_CONFIG[iZone].bPopulated THEN
                aSimHeaters[nGlobalIdx].Init(
                    rAmbient     := GVL_SimulationConfig.AMBIENT_TEMP,
                    rHeatingRate := GVL_SimulationConfig.HEATING_RATE,
                    rCoolingRate := GVL_SimulationConfig.COOLING_RATE,
                    rMaxTemp     := LREAL_TO_REAL(GVL_TemperatureZoneConfig.ZONE_CONFIG[iZone].rMaxSetpoint)
                );
            END_IF
        END_FOR
    END_FOR

    // Pressure: seed sensors with atmospheric so first-cycle reads are valid
    FOR iSensor := 1 TO GVL_PressureSystem.SENSOR_COUNT DO
        _WriteSensorRaw(
            ADR(PRG_PRESSURE_SENSOR.IO_PressureSensors[iSensor]),
            _PressureToRaw(GVL_SimulationConfig.ATMOSPHERIC_PRESSURE, iSensor));
    END_FOR

    bInitialized := TRUE;
END_METHOD

// =============================================================================
// TEMPERATURE SIMULATION
// =============================================================================

METHOD PRIVATE _SimulateTemperature
    // Channel 1: HETR_HEAD
    _SimulateElement(1,  PRG_HEAT_ZONE.HEAD_Htr,
        ADR(PRG_TEMPERATURE_SENSOR.HEAD_A),
        ADR(PRG_TEMPERATURE_SENSOR.HEAD_B));

    // Channels 2-6: A-side STR/CMB/B1/B2/B3
    _SimulateElement(2,  PRG_HEAT_ZONE.A_STR_Htr,
        ADR(PRG_TEMPERATURE_SENSOR.A_STR_A),
        ADR(PRG_TEMPERATURE_SENSOR.A_STR_B));
    _SimulateElement(3,  PRG_HEAT_ZONE.A_CMB_Htr,
        ADR(PRG_TEMPERATURE_SENSOR.A_CMB_A),
        ADR(PRG_TEMPERATURE_SENSOR.A_CMB_B));
    _SimulateElement(4,  PRG_HEAT_ZONE.A_B1_Htr,
        ADR(PRG_TEMPERATURE_SENSOR.A_B1_A),
        ADR(PRG_TEMPERATURE_SENSOR.A_B1_B));
    _SimulateElement(5,  PRG_HEAT_ZONE.A_B2_Htr,
        ADR(PRG_TEMPERATURE_SENSOR.A_B2_A),
        ADR(PRG_TEMPERATURE_SENSOR.A_B2_B));
    _SimulateElement(6,  PRG_HEAT_ZONE.A_B3_Htr,
        ADR(PRG_TEMPERATURE_SENSOR.A_B3_A),
        ADR(PRG_TEMPERATURE_SENSOR.A_B3_B));

    // Channels 7-11: B-side STR/CMB/B1/B2/B3
    _SimulateElement(7,  PRG_HEAT_ZONE.B_STR_Htr,
        ADR(PRG_TEMPERATURE_SENSOR.B_STR_A),
        ADR(PRG_TEMPERATURE_SENSOR.B_STR_B));
    _SimulateElement(8,  PRG_HEAT_ZONE.B_CMB_Htr,
        ADR(PRG_TEMPERATURE_SENSOR.B_CMB_A),
        ADR(PRG_TEMPERATURE_SENSOR.B_CMB_B));
    _SimulateElement(9,  PRG_HEAT_ZONE.B_B1_Htr,
        ADR(PRG_TEMPERATURE_SENSOR.B_B1_A),
        ADR(PRG_TEMPERATURE_SENSOR.B_B1_B));
    _SimulateElement(10, PRG_HEAT_ZONE.B_B2_Htr,
        ADR(PRG_TEMPERATURE_SENSOR.B_B2_A),
        ADR(PRG_TEMPERATURE_SENSOR.B_B2_B));
    _SimulateElement(11, PRG_HEAT_ZONE.B_B3_Htr,
        ADR(PRG_TEMPERATURE_SENSOR.B_B3_A),
        ADR(PRG_TEMPERATURE_SENSOR.B_B3_B));

    // Channels 12-13: HETR_EXH (inner + outer)
    _SimulateElement(12, PRG_HEAT_ZONE.EXH_Htr,
        ADR(PRG_TEMPERATURE_SENSOR.EXH_IN_A),
        ADR(PRG_TEMPERATURE_SENSOR.EXH_IN_B));
    _SimulateElement(13, PRG_HEAT_ZONE.EXH_E2_Htr,
        ADR(PRG_TEMPERATURE_SENSOR.EXH_OUT_A),
        ADR(PRG_TEMPERATURE_SENSOR.EXH_OUT_B));

    // Channels 14-15: HETR_CHK (inner + outer, single sensor per channel)
    _SimulateElement(14, PRG_HEAT_ZONE.CHK_Htr,
        ADR(PRG_TEMPERATURE_SENSOR.CHK_IN_A),
        0);
    _SimulateElement(15, PRG_HEAT_ZONE.CHK_E2_Htr,
        ADR(PRG_TEMPERATURE_SENSOR.CHK_OUT_A),
        0);
END_METHOD

// =============================================================================
// GAS PHYSICS SIMULATION
// =============================================================================

(* Read valve/pump states from previous cycle, run physics, produce pressures + flows *)
METHOD PRIVATE _SimulateGasPhysics
VAR
    ipOutput : I_DigitalOutput;
    ipValve  : I_Valve;
END_VAR
    // System state — null-safe (provider may transiently return 0 during init)
    ipOutput := _ipProvider.GetExhaustPump();
    fbGasPhysics.bPumpOn := (ipOutput <> 0) AND_THEN ipOutput.GetOutput();
    ipValve := _ipProvider.GetExhaustVacuumIsoValve();
    fbGasPhysics.bExhaustVacuumIsoOpen := (ipValve <> 0) AND_THEN ipValve.IsOpen();

    // Per-side valve + controller states
    fbGasPhysics.stASide := _ReadSideState(E_GasSide.A_SIDE);
    fbGasPhysics.stBSide := _ReadSideState(E_GasSide.B_SIDE);

    fbGasPhysics.Execute();
END_METHOD

(* Build ST_GasSideState from domain getters — eliminates A/B duplication.
   All provider calls are null-safe via AND_THEN to tolerate partial init. *)
METHOD PRIVATE _ReadSideState : ST_GasSideState
VAR_INPUT
    eSide : E_GasSide;
END_VAR
VAR
    ipValve  : I_Valve;
    ipCtrl   : I_Controller;
    stStatus : ST_ControllerStatus;
END_VAR
    // Gas input
    ipValve := _ipProvider.GetGasIsoValve(eSide, 1);
    _ReadSideState.bGasIsoOpen      := (ipValve <> 0) AND_THEN ipValve.IsOpen();
    ipCtrl := _ipProvider.GetMFCController(eSide);
    IF ipCtrl <> 0 THEN
        stStatus := ipCtrl.GetStatus();
        _ReadSideState.rMFCSetpoint := stStatus.rSetpoint;
    END_IF

    // Cold manifold
    ipValve := _ipProvider.GetCMBubblerValve(eSide, 1);
    _ReadSideState.bCMBubbler1Open  := (ipValve <> 0) AND_THEN ipValve.IsOpen();
    ipValve := _ipProvider.GetCMBubblerValve(eSide, 2);
    _ReadSideState.bCMBubbler2Open  := (ipValve <> 0) AND_THEN ipValve.IsOpen();
    ipValve := _ipProvider.GetCMBubblerValve(eSide, 3);
    _ReadSideState.bCMBubbler3Open  := (ipValve <> 0) AND_THEN ipValve.IsOpen();
    ipValve := _ipProvider.GetCMPurgeValve(eSide);
    _ReadSideState.bCMPurgeOpen     := (ipValve <> 0) AND_THEN ipValve.IsOpen();
    ipValve := _ipProvider.GetCMVacuumIsoValve(eSide);
    _ReadSideState.bCMVacuumIsoOpen := (ipValve <> 0) AND_THEN ipValve.IsOpen();

    // Hot manifold
    ipValve := _ipProvider.GetHMBubblerValve(eSide, 1);
    _ReadSideState.bHMBubbler1Open  := (ipValve <> 0) AND_THEN ipValve.IsOpen();
    ipValve := _ipProvider.GetHMBubblerValve(eSide, 2);
    _ReadSideState.bHMBubbler2Open  := (ipValve <> 0) AND_THEN ipValve.IsOpen();
    ipValve := _ipProvider.GetHMBubblerValve(eSide, 3);
    _ReadSideState.bHMBubbler3Open  := (ipValve <> 0) AND_THEN ipValve.IsOpen();
    ipValve := _ipProvider.GetHMPurgeValve(eSide);
    _ReadSideState.bHMPurgeOpen     := (ipValve <> 0) AND_THEN ipValve.IsOpen();
    ipValve := _ipProvider.GetHMVacuumIsoValve(eSide);
    _ReadSideState.bHMVacuumIsoOpen := (ipValve <> 0) AND_THEN ipValve.IsOpen();

    // Output
    ipValve := _ipProvider.GetNozzleIsoValve(eSide);
    _ReadSideState.bNozzleIsoOpen   := (ipValve <> 0) AND_THEN ipValve.IsOpen();
    ipCtrl := _ipProvider.GetPressureController(eSide);
    IF ipCtrl <> 0 THEN
        stStatus := ipCtrl.GetStatus();
        _ReadSideState.rPCVSetpoint := stStatus.rSetpoint;
    END_IF
END_METHOD

// =============================================================================
// PRESSURE SENSOR SIMULATION
// =============================================================================

(* Write physics-computed pressures to analog pressure sensor raw IO *)
METHOD PRIVATE _SimulatePressureSensors
    // A-side distributor (cold manifold) pressure
    _WriteSensorRaw(
        ADR(PRG_PRESSURE_SENSOR.IO_PressureSensors[E_PressureSensorIdentifier.PSNS_A_DST]),
        _PressureToRaw(LREAL_TO_REAL(fbGasPhysics.stASideOut.rCMPressure), E_PressureSensorIdentifier.PSNS_A_DST));

    // B-side distributor (cold manifold) pressure
    _WriteSensorRaw(
        ADR(PRG_PRESSURE_SENSOR.IO_PressureSensors[E_PressureSensorIdentifier.PSNS_B_DST]),
        _PressureToRaw(LREAL_TO_REAL(fbGasPhysics.stBSideOut.rCMPressure), E_PressureSensorIdentifier.PSNS_B_DST));

    // Exhaust vacuum pressure
    _WriteSensorRaw(
        ADR(PRG_PRESSURE_SENSOR.IO_PressureSensors[E_PressureSensorIdentifier.PSNS_AB_EXH]),
        _PressureToRaw(LREAL_TO_REAL(fbGasPhysics.rExhaustPressure), E_PressureSensorIdentifier.PSNS_AB_EXH));

    // Chuck vacuum pressure � driven by dedicated PUMP_CHK_VAC state
    _WriteSensorRaw(
        ADR(PRG_PRESSURE_SENSOR.IO_PressureSensors[E_PressureSensorIdentifier.PSNS_CHK_VAC]),
        _PressureToRaw(_GetChuckVacuumPressure(), E_PressureSensorIdentifier.PSNS_CHK_VAC));
END_METHOD

// =============================================================================
// MFC SIMULATION
// =============================================================================

(* Write physics-computed MFC flow to EtherCAT IO. Inert MFC uses simple ramp.
   Direct assignment to VAR members of another PROGRAM is prohibited (C0037),
   so pointer writes are used — identical pattern to _WriteSensorRaw.
   MeasuredValue is UINT (0-32000 raw counts); convert from engineering units. *)
METHOD PRIVATE _SimulateMFCs
VAR
    _pUINT : POINTER TO UINT;
END_VAR
    // A-side Precursor — from gas physics
    _pUINT := ADR(PRG_MFC.IO_MFC_Precursor.MeasuredValue);
    _pUINT^ := WORD_TO_UINT(F_EngineeringToRawCounts(
        fbGasPhysics.stASideOut.rMFCActual,
        REAL_TO_LREAL(GVL_FlowSystem.MIN_FLOW_PRECURSOR_SCCM),
        REAL_TO_LREAL(GVL_FlowSystem.MAX_FLOW_PRECURSOR_SCCM), 32000));

    // B-side Reactant — from gas physics
    _pUINT := ADR(PRG_MFC.IO_MFC_Reactant.MeasuredValue);
    _pUINT^ := WORD_TO_UINT(F_EngineeringToRawCounts(
        fbGasPhysics.stBSideOut.rMFCActual,
        REAL_TO_LREAL(GVL_FlowSystem.MIN_FLOW_REACTANT_SCCM),
        REAL_TO_LREAL(GVL_FlowSystem.MAX_FLOW_REACTANT_SCCM), 32000));

    // Inert — independent, simple ramp (not part of gas side physics)
    // CommandedSetpoint is UINT; convert to engineering units for the ramp simulator.
    fbSimMFC_Inert(
        rSetpoint := LREAL_TO_REAL(F_RawCountsToEngineering(
            PRG_MFC.IO_MFC_Inert.CommandedSetpoint,
            REAL_TO_LREAL(GVL_FlowSystem.MIN_FLOW_INERT_SCCM),
            REAL_TO_LREAL(GVL_FlowSystem.MAX_FLOW_INERT_SCCM), 32000)),
        rRampRate := GVL_SimulationConfig.MFC_RAMP_RATE
    );
    _pUINT := ADR(PRG_MFC.IO_MFC_Inert.MeasuredValue);
    _pUINT^ := WORD_TO_UINT(F_EngineeringToRawCounts(
        REAL_TO_LREAL(fbSimMFC_Inert.rActualFeedback),
        REAL_TO_LREAL(GVL_FlowSystem.MIN_FLOW_INERT_SCCM),
        REAL_TO_LREAL(GVL_FlowSystem.MAX_FLOW_INERT_SCCM), 32000));
END_METHOD

// =============================================================================
// MODBUS PRESSURE CONTROLLER SIMULATION
// =============================================================================

(* Inject physics-computed HM pressure into Modbus pressure controller adapters.
   Symmetric to PRO's EtherCAT path which writes IO_CtrlASide.MeasuredValue directly:
   InjectMeasuredValue() overwrites the value that Modbus polling would normally update. *)
METHOD PRIVATE _SimulateModbusPressureControllers
    PRG_BronkhorstPressure.aDrivers[E_PressureController.A_Side].InjectMeasuredValue(fbGasPhysics.stASideOut.rHMPressure);
    PRG_BronkhorstPressure.aDrivers[E_PressureController.B_Side].InjectMeasuredValue(fbGasPhysics.stBSideOut.rHMPressure);
END_METHOD

// =============================================================================
// PRIVATE HELPERS
// =============================================================================

(* Run physics for one channel and write result to both A+B redundant sensor channels *)
METHOD PRIVATE _SimulateElement
VAR_INPUT
    nGlobalIdx : INT;
    bHeaterOn  : BOOL;
    pSensorA   : POINTER TO BYTE;
    pSensorB   : POINTER TO BYTE;
END_VAR
VAR
    nRawValue : INT;
END_VAR
    IF nGlobalIdx < 1 OR nGlobalIdx > GVL_TemperatureZones.CHANNEL_MAX THEN RETURN; END_IF
    aSimHeaters[nGlobalIdx](bHeaterOn := bHeaterOn);
    nRawValue := _TempToRaw(aSimHeaters[nGlobalIdx].rCurrentTemp);
    _WriteSensorRaw(pSensorA, nRawValue);
    _WriteSensorRaw(pSensorB, nRawValue);
END_METHOD

(* Return the simulated chuck vacuum pressure based on PUMP_CHK_VAC output state.
   PUMP_CHK_VAC is the dedicated chuck vacuum pump (not shared with exhaust).
   Pump ON  ? vacuum achieved: CHUCK_VACUUM_PRESSURE (0.01 bar)
   Pump OFF ? atmospheric: ATMOSPHERIC_PRESSURE (1.0 bar) *)
METHOD PRIVATE _GetChuckVacuumPressure : REAL
VAR
    ipPump : I_DigitalOutput;
END_VAR
    ipPump := _ipProvider.GetDigitalOutput(E_DigitalOutputIdentifier.PUMP_CHK_VAC);
    _GetChuckVacuumPressure := SEL(
        (ipPump <> 0) AND_THEN ipPump.GetOutput(),
        GVL_SimulationConfig.ATMOSPHERIC_PRESSURE,
        GVL_SimulationConfig.CHUCK_VACUUM_PRESSURE);
END_METHOD

(* Convert °C to Beckhoff EL32xx raw INT. Scale: 0.1°C per count → 25.0°C = 250 *)
METHOD PRIVATE _TempToRaw : INT
VAR_INPUT
    rTempC : REAL;
END_VAR
    _TempToRaw := REAL_TO_INT(rTempC / LREAL_TO_REAL(GVL_TemperatureSystem.SCALE_BECKHOFF_TEMP));
END_METHOD

(* Convert bar to Beckhoff EL3048 raw INT using per-sensor scaling from GVL_PressureSystem.
   Each sensor has different raw/scaled ranges. *)
METHOD PRIVATE _PressureToRaw : INT
VAR_INPUT
    rBar     : REAL;
    nSensor  : INT;
END_VAR
    CASE nSensor OF
    1: // PSNS_A_DST: 0-30518 raw → 0-3 bar
        _PressureToRaw := F_ScaleRealToInt(rBar,
            LREAL_TO_REAL(GVL_PressureSystem.PSNS_A_DST_SCALED_MIN),
            LREAL_TO_REAL(GVL_PressureSystem.PSNS_A_DST_SCALED_MAX),
            LREAL_TO_INT(GVL_PressureSystem.PSNS_A_DST_RAW_MIN),
            LREAL_TO_INT(GVL_PressureSystem.PSNS_A_DST_RAW_MAX));
    2: // PSNS_B_DST: 0-30518 raw → 0-3 bar
        _PressureToRaw := F_ScaleRealToInt(rBar,
            LREAL_TO_REAL(GVL_PressureSystem.PSNS_B_DST_SCALED_MIN),
            LREAL_TO_REAL(GVL_PressureSystem.PSNS_B_DST_SCALED_MAX),
            LREAL_TO_INT(GVL_PressureSystem.PSNS_B_DST_RAW_MIN),
            LREAL_TO_INT(GVL_PressureSystem.PSNS_B_DST_RAW_MAX));
    3: // PSNS_AB_EXH: 0-30518 raw → 0-1 bar
        _PressureToRaw := F_ScaleRealToInt(rBar,
            LREAL_TO_REAL(GVL_PressureSystem.PSNS_AB_EXH_SCALED_MIN),
            LREAL_TO_REAL(GVL_PressureSystem.PSNS_AB_EXH_SCALED_MAX),
            LREAL_TO_INT(GVL_PressureSystem.PSNS_AB_EXH_RAW_MIN),
            LREAL_TO_INT(GVL_PressureSystem.PSNS_AB_EXH_RAW_MAX));
    4: // PSNS_CHK_VAC: 3052-15259 raw → 0.00325-1.01325 bar (inverted physical)
        _PressureToRaw := F_ScaleRealToInt(rBar,
            LREAL_TO_REAL(GVL_PressureSystem.PSNS_CHK_VAC_SCALED_MIN),
            LREAL_TO_REAL(GVL_PressureSystem.PSNS_CHK_VAC_SCALED_MAX),
            LREAL_TO_INT(GVL_PressureSystem.PSNS_CHK_VAC_RAW_MIN),
            LREAL_TO_INT(GVL_PressureSystem.PSNS_CHK_VAC_RAW_MAX));
    END_CASE
END_METHOD

(* Write raw INT to a Beckhoff sensor struct at offset 2.
   All EL3xxx structs share the same memory layout:
   Offset 0-1: Status WORD, Offset 2-3: Value INT.
   This matches how FB_AnalogInputAdapter reads — same offset, reverse direction. *)
METHOD PRIVATE _WriteSensorRaw
VAR_INPUT
    pSensor   : POINTER TO BYTE;
    nRawValue : INT;
END_VAR
VAR
    pValue : POINTER TO INT;
END_VAR
    IF pSensor = 0 THEN RETURN; END_IF
    pValue := pSensor + 2;
    pValue^ := nRawValue;
END_METHOD

END_PROGRAM

(* ---- PRG_Spectrometer.st ---- *)
(*
PRG_Spectrometer — Runs the spectrometer hardware driver at 1ms cycle.
*)
PROGRAM PRG_Spectrometer
VAR
    stOutputRegisters      AT%Q* : ST_OutputRegistersRaw;
    stInputRegisters       AT%I* : ST_InputRegistersRaw;
    aInputLogicSignals     AT%I* : ARRAY[1..4] OF USINT;
    aOutputLogicSignals    AT%Q* : ARRAY[1..4] OF USINT;
    fbSpectrometer               : FB_Spectrometer;
    stTelemetry                  : ST_SpectrometerTelemetryData;
    stDebugControls              : ST_DebugControls;
    _bInitialized                : BOOL := FALSE;
END_VAR

    IF NOT _bInitialized THEN
        _bInitialized := fbSpectrometer.Init(
            refOutput             := stOutputRegisters,
            refInput              := stInputRegisters,
            refInputLogicSignals  := aInputLogicSignals,
            refOutputLogicSignals := aOutputLogicSignals
        );
    END_IF

    IF NOT _bInitialized THEN
        RETURN;
    END_IF

    // 1. Execute hardware handshake (STROBE/ACK)
    fbSpectrometer.Execute();

    // 2. Publish telemetry (read by DALP Manager via ADS at 1ms)
    stTelemetry.Measurement := fbSpectrometer.GetMeasurement();
    stTelemetry.Settings    := fbSpectrometer.GetDeviceSettings();

    // 3. Manual debug overrides
    IF stDebugControls.bApplyLimits THEN
        fbSpectrometer.SetSpectrumLimits(
            nStartRatio  := stDebugControls.StartRatio,
            nStopRatio   := stDebugControls.StopRatio,
            nTotalPixels := stDebugControls.nTotalPixels
        );
        stDebugControls.bApplyLimits := FALSE;
    END_IF

    IF stDebugControls.bApplyFreq THEN
        fbSpectrometer.SetFrequency(ScanRate := TO_UDINT(stDebugControls.Frequency));
        stDebugControls.bApplyFreq := FALSE;
    END_IF

    IF stDebugControls.bApplyLight THEN
        fbSpectrometer.SetLightIntensity(
            TargetLight := stDebugControls.TargetLight,
            AutoAdjust  := TRUE
        );
        stDebugControls.bApplyLight := FALSE;
    END_IF

END_PROGRAM

(* ---- PRG_Telemetry.st ---- *)
(*
PRG_Telemetry — Orchestrates telemetry publication and command dispatch.
Called every scan from PRG_SHARK after all subsystems have been updated.

Publishes the detailed (per-channel) telemetry view from the subsystem
references.

ADS Symbol Mapping:
  READ:  PRG_Telemetry.fbTelemetryPublisher.stTelemetry               (ST_MachineTelemetry)
  WRITE: PRG_Telemetry.fbCommandReceiver.AdsStream                    (ARRAY[0..4095] OF BYTE)
  READ:  PRG_Telemetry.fbCommandReceiver.nLastCommandIndex            (DINT)
*)
PROGRAM PRG_Telemetry
VAR
    fbTelemetryPublisher        : FB_TelemetryPublisher;
    fbCommandReceiver           : FB_CommandReceiver;
    _bInitialized               : BOOL := FALSE;
END_VAR

    IF NOT _bInitialized THEN
        _Init();
        RETURN;
    END_IF

    _Execute();

METHOD PRIVATE _Init
VAR
    bOk : BOOL;
END_VAR
    bOk := fbTelemetryPublisher.Init(
        refValveSub    := PRG_VALVE.fbValveSubsystem,
        refFlowSub     := PRG_MFC.fbFlowSubsystem,
        refPressureSub := PRG_PRESSURE_SENSOR.fbPressureSubsystem,
        refTempSub     := PRG_HEAT_ZONE.fbTemperatureSubsystem,
        refDISub       := PRG_DIGITAL_INPUT.fbDigitalInputSubsystem,
        refDOSub       := PRG_DIGITAL_OUTPUT.fbDigitalOutputSubsystem
    );
    IF NOT bOk THEN RETURN; END_IF

    bOk := fbCommandReceiver.Init(
        ipHardware            := PRG_SHARK.fbHardwareProvider,
        ipSpectrometer        := PRG_Spectrometer.fbSpectrometer,
        rTempDisableThreshold := 0.0,
        refOrchestrator       := PRG_Sequence.fbOrchestrator
    );
    IF NOT bOk THEN RETURN; END_IF

    _bInitialized := TRUE;
END_METHOD

METHOD PRIVATE _Execute
    // Update telemetry struct (read by clients via ADS)
    fbTelemetryPublisher();

    // Poll for incoming commands (written by clients via ADS)
    fbCommandReceiver();

    // Echo last command index into the telemetry struct for client-side sync
    fbTelemetryPublisher.SetCommandIndex(nCommandIndex := fbCommandReceiver.nLastCommandIndex);
END_METHOD

END_PROGRAM

(* ---- PRG_TEMPERATURE_SENSOR.st ---- *)
PROGRAM PRG_TEMPERATURE_SENSOR
(*
Shark temperature sensor wiring program.

  * 10 channels total (one per RTD+SSR pair) split across 8 zones.
  * Each channel keeps its existing A+B redundant RTDs wrapped in
    FB_DualSensor; the resulting I_Sensor is what the channel controller sees.
  * Channel ordering MUST match the order zones appear in E_HeatZone
    times the order channels appear within each zone. The subsystem
    relies on this ordering when slicing the flat channel array per zone.

Channel layout:
  HETR_HEAD   (1)      Shared head
  HETR_A_STR  (2)      A-side start (umbilical)
  HETR_A_CMB  (3)      A-side combiner / hot manifold
  HETR_A_B1   (4)      A-side bubbler 1
  HETR_A_B2   (5)      A-side bubbler 2
  HETR_A_B3   (6)      A-side bubbler 3
  HETR_B_STR  (7)      B-side start (umbilical)
  HETR_B_CMB  (8)      B-side combiner / hot manifold
  HETR_B_B1   (9)      B-side bubbler 1
  HETR_B_B2   (10)     B-side bubbler 2
  HETR_B_B3   (11)     B-side bubbler 3
  HETR_EXH    (12..13) Exhaust inner, outer
  HETR_CHK    (14..15) Chuck inner, outer
*)
VAR
    // --- Hardware IO (linked to EtherCAT process image) ---

    // HETR_HEAD (channel 1)
    HEAD_A   : T_Beckhoff_TempSensor_General;   // 1
    HEAD_B   : T_Beckhoff_TempSensor_General;   // 2
    // HETR_A_STR (channel 2)
    A_STR_A  : T_Beckhoff_TempSensor_General;   // 3
    A_STR_B  : T_Beckhoff_TempSensor_General;   // 4
    // HETR_A_CMB (channel 3)
    A_CMB_A  : T_Beckhoff_TempSensor_General;   // 5
    A_CMB_B  : T_Beckhoff_TempSensor_General;   // 6
    // HETR_A_B1 (channel 4)
    A_B1_A   : T_Beckhoff_TempSensor_General;   // 7
    A_B1_B   : T_Beckhoff_TempSensor_General;   // 8
    // HETR_A_B2 (channel 5)
    A_B2_A   : T_Beckhoff_TempSensor_General;   // 9
    A_B2_B   : T_Beckhoff_TempSensor_General;   // 10
    // HETR_A_B3 (channel 6)
    A_B3_A   : T_Beckhoff_TempSensor_General;   // 11
    A_B3_B   : T_Beckhoff_TempSensor_General;   // 12
    // HETR_B_STR (channel 7)
    B_STR_A  : T_Beckhoff_TempSensor_General;   // 13
    B_STR_B  : T_Beckhoff_TempSensor_General;   // 14
    // HETR_B_CMB (channel 8)
    B_CMB_A  : T_Beckhoff_TempSensor_General;   // 15
    B_CMB_B  : T_Beckhoff_TempSensor_General;   // 16
    // HETR_B_B1 (channel 9)
    B_B1_A   : T_Beckhoff_TempSensor_General;   // 17
    B_B1_B   : T_Beckhoff_TempSensor_General;   // 18
    // HETR_B_B2 (channel 10)
    B_B2_A   : T_Beckhoff_TempSensor_General;   // 19
    B_B2_B   : T_Beckhoff_TempSensor_General;   // 20
    // HETR_B_B3 (channel 11)
    B_B3_A   : T_Beckhoff_TempSensor_General;   // 21
    B_B3_B   : T_Beckhoff_TempSensor_General;   // 22
    // HETR_EXH (channels 12..13)
    EXH_IN_A    : T_Beckhoff_TempSensor_General;   // 23
    EXH_IN_B    : T_Beckhoff_TempSensor_General;   // 24
    EXH_OUT_A    : T_Beckhoff_TempSensor_General;   // 25
    EXH_OUT_B    : T_Beckhoff_TempSensor_General;   // 26
    // HETR_CHK (channels 14..15) — single sensor per channel (A only)
    CHK_IN_A    : T_Beckhoff_TempSensor_Chuck;     // 27
    CHK_OUT_A    : T_Beckhoff_TempSensor_Chuck;    // 28

    // Stage temperature sensors (monitor only — no heater/PID)
    STG_X_TEMP  : T_Beckhoff_TempSensor_General;   // SENS_STAGE_X (2) — Stage X-axis temperature
    STG_Y_TEMP  : T_Beckhoff_TempSensor_General;   // SENS_STAGE_Y (3) — Stage Y-axis temperature
    AMBT_TEMP   : T_Beckhoff_AmbientSensor;         // SENS_CHAMBER (1) — TH sensor temperature channel
    SIDE_A_TEMP : T_Beckhoff_TempSensor_General;    // SENS_A_SIDE  (4) — A-side temperature
    SIDE_B_TEMP : T_Beckhoff_TempSensor_General;    // SENS_B_SIDE  (5) — B-side temperature

    // --- Monitor sensor FBs (one adapter+sensor per monitor zone) ---
    fbChamberAdapter  : FB_AnalogInputAdapter;  // SENS_CHAMBER (1)
    fbChamberSensor   : FB_AnalogSensor;
    fbStgXAdapter     : FB_AnalogInputAdapter;  // SENS_STAGE_X (2)
    fbStgXSensor      : FB_AnalogSensor;
    fbStgYAdapter     : FB_AnalogInputAdapter;  // SENS_STAGE_Y (3)
    fbStgYSensor      : FB_AnalogSensor;
    fbSideAAdapter    : FB_AnalogInputAdapter;  // SENS_A_SIDE  (4)
    fbSideASensor     : FB_AnalogSensor;
    fbSideBAdapter    : FB_AnalogInputAdapter;  // SENS_B_SIDE  (5)
    fbSideBSensor     : FB_AnalogSensor;

    // --- Adapters & Sensors (one A+B pair per channel) ---
    afbAdapters_A   : ARRAY[1..GVL_TemperatureZones.CHANNEL_MAX] OF FB_AnalogInputAdapter;
    afbAdapters_B   : ARRAY[1..GVL_TemperatureZones.CHANNEL_MAX] OF FB_AnalogInputAdapter;
    afbSensors_A    : ARRAY[1..GVL_TemperatureZones.CHANNEL_MAX] OF FB_AnalogSensor;    // EXH: channels 12..13; CHK: channels 14..15
    afbSensors_B    : ARRAY[1..GVL_TemperatureZones.CHANNEL_MAX] OF FB_AnalogSensor;
    afbDualSensors  : ARRAY[1..GVL_TemperatureZones.CHANNEL_MAX] OF FB_DualSensor;
    _abHasChannelB  : ARRAY[1..GVL_TemperatureZones.CHANNEL_MAX] OF BOOL;  // FALSE for single-sensor channels (e.g. CHK) — their B adapter/sensor are never initialized and must not be executed

    // --- Interface arrays consumed by FB_TemperatureSubsystem ---
    aipChannelSensors : ARRAY[1..GVL_TemperatureZones.CHANNEL_MAX] OF I_Sensor;
    aipMonitorSensors : ARRAY[1..GVL_TemperatureZones.MONITOR_ZONE_COUNT] OF I_Sensor;  // 1=SENS_CHAMBER, 2=SENS_STAGE_X, 3=SENS_STAGE_Y, 4=SENS_A_SIDE, 5=SENS_B_SIDE

    bInitialized : BOOL := FALSE;
    i : INT;
END_VAR

    IF NOT bInitialized THEN
        _Init();
    END_IF

    // Execute every channel's A + B + dual composite.
    // Single-sensor channels (B pointer null at init) have no B adapter/sensor —
    // skip them, otherwise the never-initialized B FB raises 'Sensor not
    // initialized' (with an empty source) on every scan cycle.
    FOR i := 1 TO GVL_TemperatureZones.CHANNEL_MAX DO
        afbAdapters_A[i].Execute();
        afbSensors_A[i].Execute();
        IF _abHasChannelB[i] THEN
            afbAdapters_B[i].Execute();
            afbSensors_B[i].Execute();
        END_IF
        afbDualSensors[i].Execute();
    END_FOR

    // Execute monitor sensors (one adapter+sensor pair per zone)
    fbChamberAdapter.Execute();  fbChamberSensor.Execute();
    fbStgXAdapter.Execute();     fbStgXSensor.Execute();
    fbStgYAdapter.Execute();     fbStgYSensor.Execute();
    fbSideAAdapter.Execute();    fbSideASensor.Execute();
    fbSideBAdapter.Execute();    fbSideBSensor.Execute();

METHOD PRIVATE _Init
    // Wire each channel's A+B raw RTDs into a dual sensor.
    // Order MUST match the channel layout in the file header.
    _InitElement(1,  ADR(HEAD_A),  ADR(HEAD_B));
    _InitElement(2,  ADR(A_STR_A), ADR(A_STR_B));
    _InitElement(3,  ADR(A_CMB_A), ADR(A_CMB_B));
    _InitElement(4,  ADR(A_B1_A),  ADR(A_B1_B));
    _InitElement(5,  ADR(A_B2_A),  ADR(A_B2_B));
    _InitElement(6,  ADR(A_B3_A),  ADR(A_B3_B));
    _InitElement(7,  ADR(B_STR_A), ADR(B_STR_B));
    _InitElement(8,  ADR(B_CMB_A), ADR(B_CMB_B));
    _InitElement(9,  ADR(B_B1_A),  ADR(B_B1_B));
    _InitElement(10, ADR(B_B2_A),  ADR(B_B2_B));
    _InitElement(11, ADR(B_B3_A),  ADR(B_B3_B));
    _InitElement(12, ADR(EXH_IN_A),   ADR(EXH_IN_B));      // EXH: Inner
    _InitElement(13, ADR(EXH_OUT_A),   ADR(EXH_OUT_B));     // EXH: Outer
    _InitElement(14, ADR(CHK_IN_A),    0);          // CHK: single sensor per channel
    _InitElement(15, ADR(CHK_OUT_A),   0);          // CHK: single sensor per channel

    // Wire monitor sensors (one per E_TemperatureMonitorZone entry)
    _InitMonitorSensor(
        eZone      := E_TemperatureMonitorZone.SENS_CHAMBER,
        sName      := 'AMBT_TEMP',
        refAdapter := fbChamberAdapter,
        refSensor  := fbChamberSensor,
        pChannel   := ADR(AMBT_TEMP),
        rRawMin    := GVL_TemperatureSystem.AMBT_TEMP_RAW_MIN,
        rRawMax    := GVL_TemperatureSystem.AMBT_TEMP_RAW_MAX,
        rScaledMin := GVL_TemperatureSystem.AMBT_TEMP_SCALED_MIN,
        rScaledMax := GVL_TemperatureSystem.AMBT_TEMP_SCALED_MAX
    );
    _InitMonitorSensor(
        eZone      := E_TemperatureMonitorZone.SENS_STAGE_X,
        sName      := 'STG_X_TEMP',
        refAdapter := fbStgXAdapter,
        refSensor  := fbStgXSensor,
        pChannel   := ADR(STG_X_TEMP),
        rRawMin    := 0.0,
        rRawMax    := GVL_TemperatureSystem.TEMP_RAW_AT_MAX_SENSOR,
        rScaledMin := 0.0,
        rScaledMax := GVL_TemperatureSystem.SENSOR_MAX_TEMP
    );
    _InitMonitorSensor(
        eZone      := E_TemperatureMonitorZone.SENS_STAGE_Y,
        sName      := 'STG_Y_TEMP',
        refAdapter := fbStgYAdapter,
        refSensor  := fbStgYSensor,
        pChannel   := ADR(STG_Y_TEMP),
        rRawMin    := 0.0,
        rRawMax    := GVL_TemperatureSystem.TEMP_RAW_AT_MAX_SENSOR,
        rScaledMin := 0.0,
        rScaledMax := GVL_TemperatureSystem.SENSOR_MAX_TEMP
    );
    _InitMonitorSensor(
        eZone      := E_TemperatureMonitorZone.SENS_A_SIDE,
        sName      := 'SIDE_A_TEMP',
        refAdapter := fbSideAAdapter,
        refSensor  := fbSideASensor,
        pChannel   := ADR(SIDE_A_TEMP),
        rRawMin    := 0.0,
        rRawMax    := GVL_TemperatureSystem.TEMP_RAW_AT_MAX_SENSOR,
        rScaledMin := 0.0,
        rScaledMax := GVL_TemperatureSystem.SENSOR_MAX_TEMP
    );
    _InitMonitorSensor(
        eZone      := E_TemperatureMonitorZone.SENS_B_SIDE,
        sName      := 'SIDE_B_TEMP',
        refAdapter := fbSideBAdapter,
        refSensor  := fbSideBSensor,
        pChannel   := ADR(SIDE_B_TEMP),
        rRawMin    := 0.0,
        rRawMax    := GVL_TemperatureSystem.TEMP_RAW_AT_MAX_SENSOR,
        rScaledMin := 0.0,
        rScaledMax := GVL_TemperatureSystem.SENSOR_MAX_TEMP
    );

    bInitialized := TRUE;
END_METHOD

METHOD PRIVATE _InitElement
VAR_INPUT
    nGlobalIdx : INT;
    pChannel_A : POINTER TO BYTE;
    pChannel_B : POINTER TO BYTE;  // NULL (0) for single-sensor channels
END_VAR
VAR
    ipSecondary : I_Sensor;  // NULL when pChannel_B is null (triggers FB_DualSensor single-mode)
END_VAR
    // Channel A (always present)
    afbAdapters_A[nGlobalIdx].Link(pChannel_A);
    afbSensors_A[nGlobalIdx].Init(
        sInstanceName := CONCAT('TEMP_E', CONCAT(TO_STRING(nGlobalIdx), '_A')),
        ipRawInput    := afbAdapters_A[nGlobalIdx],
        rRawMin       := 0.0,
        rRawMax       := GVL_TemperatureSystem.TEMP_RAW_AT_MAX_SENSOR,
        rScaledMin    := 0.0,
        rScaledMax    := GVL_TemperatureSystem.SENSOR_MAX_TEMP
    );

    // Channel B (optional - skip if null pointer provided)
    IF pChannel_B <> 0 THEN
        afbAdapters_B[nGlobalIdx].Link(pChannel_B);
        afbSensors_B[nGlobalIdx].Init(
            sInstanceName := CONCAT('TEMP_E', CONCAT(TO_STRING(nGlobalIdx), '_B')),
            ipRawInput    := afbAdapters_B[nGlobalIdx],
            rRawMin       := 0.0,
            rRawMax       := GVL_TemperatureSystem.TEMP_RAW_AT_MAX_SENSOR,
            rScaledMin    := 0.0,
            rScaledMax    := GVL_TemperatureSystem.SENSOR_MAX_TEMP
        );
        ipSecondary := afbSensors_B[nGlobalIdx];
        _abHasChannelB[nGlobalIdx] := TRUE;
    ELSE
        // Single-sensor mode: secondary remains NULL, triggering FB_DualSensor single-mode
        ipSecondary := 0;
        _abHasChannelB[nGlobalIdx] := FALSE;
    END_IF

    // Dual composite (single-mode when ipSecondary = 0)
    afbDualSensors[nGlobalIdx].Init(
        sInstanceName := CONCAT('DUAL_E', TO_STRING(nGlobalIdx)),
        ipPrimary     := afbSensors_A[nGlobalIdx],
        ipSecondary   := ipSecondary,
        rMaxDeviation := GVL_TemperatureZoneConfig.CHANNEL_MAX_DEVIATION[nGlobalIdx]
    );
    aipChannelSensors[nGlobalIdx] := afbDualSensors[nGlobalIdx];
END_METHOD

METHOD PRIVATE _InitMonitorSensor
VAR_INPUT
    eZone      : E_TemperatureMonitorZone;
    sName      : STRING;
    pChannel   : POINTER TO BYTE;
    rRawMin    : LREAL;
    rRawMax    : LREAL;
    rScaledMin : LREAL;
    rScaledMax : LREAL;
END_VAR
VAR_IN_OUT
    refAdapter : FB_AnalogInputAdapter;
    refSensor  : FB_AnalogSensor;
END_VAR
    refAdapter.Link(pChannel);
    refSensor.Init(
        sInstanceName := sName,
        ipRawInput    := refAdapter,
        rRawMin       := rRawMin,
        rRawMax       := rRawMax,
        rScaledMin    := rScaledMin,
        rScaledMax    := rScaledMax
    );
    aipMonitorSensors[eZone] := refSensor;
END_METHOD

END_PROGRAM

(* ---- PRG_VALVE.st ---- *)
(*
Valve Program - Shark System
1 SMC block (4 bytes) for 29 pneumatic valves (1-29).
6 solenoid valves (30-35) via injected I_DigitalOutput from PRG_DIGITAL_OUTPUT.
*)
PROGRAM PRG_VALVE
VAR
    // Subsystem and Manual Panel
    fbValveSubsystem : FB_ValveSubsystem;
    fbManualPanel    : FB_ValveManualPanel;

    // SMC EtherCAT Output Block (1 block, 4 bytes = 32 bits, uses bits 0-28)
    IO_SMC_Outputs AT %Q* : ARRAY[0..3] OF BYTE;
    fbSMC : FB_SMCOutputBlock;

    // SMC Adapters for Pneumatic Valves (1-29)
    afbSMCAdapters : ARRAY[1..GVL_ValveSystem.PNEUMATIC_VALVE_COUNT] OF FB_SMCAdapter;

    // Universal Valve Array
    afbValves : ARRAY[1..GVL_ValveSystem.VALVE_COUNT] OF FB_Valve;
    aipValves : ARRAY[1..GVL_ValveSystem.VALVE_COUNT] OF I_Valve;

    // Injected interfaces for solenoid valves (30-35)
    _ipChuckLZ1  : I_DigitalOutput;
    _ipChuckLZ2  : I_DigitalOutput;
    _ipChuckLZ3  : I_DigitalOutput;
    _ipChuckVent : I_DigitalOutput;
    _ipChuckWIn  : I_DigitalOutput;
    _ipChuckWOut : I_DigitalOutput;

    bConfigured     : BOOL := FALSE;
    bInitialized    : BOOL := FALSE;
    _bNotConfiguredLogged : BOOL := FALSE;
    i : INT;
END_VAR

    IF NOT bConfigured THEN
        IF NOT _bNotConfiguredLogged THEN
            GVL_ErrorLogger.Logger.LogError(
                sSource  := 'PRG_VALVE',
                eErrorId := E_ErrorId.ERR_GEN_NOT_CONFIGURED,
                sContext := 'PRG_VALVE executed before Configure(); valve program will not run'
            );
            _bNotConfiguredLogged := TRUE;
        END_IF
        RETURN;
    END_IF

    IF NOT bInitialized THEN
        _Init();
    END_IF

    // Execute SMC block
    fbSMC(aOutputBytes := IO_SMC_Outputs);

    // Execute valve logic
    FOR i := 1 TO GVL_ValveSystem.VALVE_COUNT DO
        afbValves[i].Execute();
    END_FOR

    // Update subsystem status
    fbValveSubsystem.Execute();
    fbManualPanel(ipSubsystem := fbValveSubsystem, nMaxValveId := GVL_ValveSystem.VALVE_COUNT);

METHOD PUBLIC Configure
VAR_INPUT
    ipChuckLZ1  : I_DigitalOutput;
    ipChuckLZ2  : I_DigitalOutput;
    ipChuckLZ3  : I_DigitalOutput;
    ipChuckVent : I_DigitalOutput;
    ipChuckWIn  : I_DigitalOutput;
    ipChuckWOut : I_DigitalOutput;
END_VAR
    IF bConfigured THEN RETURN;
    END_IF

    _ipChuckLZ1  := ipChuckLZ1;
    _ipChuckLZ2  := ipChuckLZ2;
    _ipChuckLZ3  := ipChuckLZ3;
    _ipChuckVent := ipChuckVent;
    _ipChuckWIn  := ipChuckWIn;
    _ipChuckWOut := ipChuckWOut;

    bConfigured := TRUE;
END_METHOD

METHOD PRIVATE _Init
VAR
    iLocal   : INT;
END_VAR
    // Default: leave all valves unbound
    FOR iLocal := 1 TO GVL_ValveSystem.VALVE_COUNT DO
        aipValves[iLocal] := 0;
    END_FOR

    // Execute SMC block once to capture byte-array address, then clear
    fbSMC(aOutputBytes := IO_SMC_Outputs);
    fbSMC.ClearAll();

    // Initialize Pneumatic Valves (1-29) on SMC Block
    FOR iLocal := 1 TO GVL_ValveSystem.PNEUMATIC_VALVE_COUNT DO
        afbSMCAdapters[iLocal].Init(refBlock := fbSMC, nIndex := INT_TO_USINT(iLocal - 1));
        afbValves[iLocal].Init(sInstanceName := INT_TO_STRING(iLocal), ipOutput := afbSMCAdapters[iLocal]);
        aipValves[iLocal] := afbValves[iLocal];
    END_FOR

    // Initialize Solenoid Valves (30-35) using injected digital outputs
    _InitInjectedValve(E_ValveIdentifier.VALV_CHK_LZ1,  _ipChuckLZ1);
    _InitInjectedValve(E_ValveIdentifier.VALV_CHK_LZ2,  _ipChuckLZ2);
    _InitInjectedValve(E_ValveIdentifier.VALV_CHK_LZ3,  _ipChuckLZ3);
    _InitInjectedValve(E_ValveIdentifier.VALV_CHK_VENT, _ipChuckVent);
    _InitInjectedValve(E_ValveIdentifier.VALV_CHK_WIN,  _ipChuckWIn);
    _InitInjectedValve(E_ValveIdentifier.VALV_CHK_WOUT, _ipChuckWOut);

    fbValveSubsystem.Init(aipValves := aipValves, nCount := GVL_ValveSystem.VALVE_COUNT);
    bInitialized := TRUE;
END_METHOD

METHOD PRIVATE _InitInjectedValve
VAR_INPUT
    eValve   : E_ValveIdentifier;
    ipOutput : I_DigitalOutput;
END_VAR
    IF ipOutput = 0 THEN RETURN; END_IF

    afbValves[eValve].Init(sInstanceName := TO_STRING(eValve), ipOutput := ipOutput);
    aipValves[eValve] := afbValves[eValve];
END_METHOD

END_PROGRAM
